FUNCTION F_PartPickupSuccess : BOOL
VAR_INPUT
	WX : sBogie;
END_VAR
VAR
END_VAR

IF WX.bEnabled THEN
	IF WX.A.bClamped AND WX.B.bClamped AND F_PartIsPresent(WX) AND WX.ConveyorLoadPos = 0 THEN
		
		F_PartPickupSuccess := 1;
 
	ELSE
		F_PartPickupSuccess := 0;
		RETURN;
	END_IF
	
	RETURN;
	
END_IF

END_FUNCTION

(* stored: Version 1.1.0.1, ProductVersion 3.1.4024.12
   POU F_PartPickupSuccess: Id {93365b99-2d8f-4328-a255-2a51dc0adb9a}, SpecialFunc None *)
